(* Logix 5000 project; controller BTS01 vendor 1 type 14 code 217 rev 32.14; software revision 32.04; part 14 of 15 *)
(* tags used below, declared in another part *)
   AG1101 : DTE_VFD;   // Tank 1100 Agitator
   AG1101_CIP_ENABLE : BOOL;
   AG1101_ONS : DINT;
   AG1201 : DTE_VFD;   // Tank 1200 Agitator
   AG1201_CIP_ENABLE : BOOL;
   AG1201_ONS : DINT;
   AirblowPB : BOOL;
   C02S01 : REAL[8];   // 5069-IF8
   C02S02 : REAL[8];   // 5069-OF8
   C02S03 : INT;   // 5069-IB16
   C02S05 : INT;   // 5069-OB16
   C02S06 : INT;   // 5069-IB16
   CIP_1_ACTIVE_CIRCUIT : DINT;
   CIP_1_CIRCUIT_SELECT_HMI : INT;
   CIP_1_RUN_LATCH : BOOL;
   CIP_1_SEQ_CTU : COUNTER;   // CIP 1 SEQUENCE STEP COUNTER THIS IS THE SEQUENCE STEP CONTROL
   CIP_Circuit_1_Visibility : BOOL;
   CIP_Circuit_2_Visibility : BOOL;
   CIP_Circuit_3_Visibility : BOOL;
   CIP_Circuit_4_Visibility : BOOL;
   CIP_SUPPLY_PUMP_CIP_ENABLE : BOOL;
   FP1000_CIP_Supply_Ind : DINT;
   FP1001_CIP_Return_Ind : DINT;
   GlobalAlmAck : BOOL;
   HMIAlarms : DINT[25];   // Alarm Trigger Array
   ONS : DINT[20];   // ONE_SHOT_BIT
   P1001 : DTE_VFD;   // Dressing Tank Fill Pump
   P1001_CIP_Enable : BOOL;
   P1001_ONS : DINT;
   P1001_Start_Request : BOOL;
   P1002 : DTE_VFD;   // Product Filler Fill Pump
   P1002_CIP_ENABLE : BOOL;
   P1002_ONS : DINT;
   P1003 : DTE_VFD;   // CIP Return Pump
   P1003_CIP_ENABLE : BOOL;
   P1003_ONS : DINT;
   P1003_Start_Delay_TMR1 : TIMER;   // CIP Return Pump Active CIP Circuit 1 Start Delay Timer
   P1003_Start_Delay_TMR2 : TIMER;   // CIP Return Pump Active CIP Circuit 2 Start Delay Timer
   P1004 : DTE_VFD;   // Filler CIP Return Pump
   P1004_ONS : DINT;
   TransferEnabled : BOOL;
   TransferSelected : DINT;
   TransferSelection : DINT;
   TransferStandby : BOOL;
   TransferStartPB : BOOL;
   TransferStartPBTimer : TIMER;
   TransferStartPBVisibility : BOOL;
   TransferStopPB : BOOL;
   UnloadEnabled : BOOL;
   UnloadSelected : DINT;
   UnloadSelection : DINT;
   UnloadStandby : BOOL;
   UnloadStartPB : BOOL;
   UnloadStartPBTimer : TIMER;
   UnloadStartPBVisibility : BOOL;
   UnloadStopPB : BOOL;
   V1101 : DTE_Air_Valve_v2;   // Tank 1100 Fill Valve
   V1201 : DTE_Air_Valve_v2;   // Tank 1200 Fill Valve
   ZS1000_1_Ind : DINT;
   ZS1000_2_Ind : DINT;
   ZS1000_3_Ind : DINT;
   ZS1000_4_Ind : DINT;
   ZS1000_5_Ind : DINT;
   ZS1001_1_Ind : DINT;
   ZS1001_2_Ind : DINT;
   ZS1001_3_Ind : DINT;
   ZS1001_4_Ind : DINT;
   ZS1001_5_Ind : DINT;
   ZS1101_Ind : DINT;
   ZS1201_Ind : DINT;
(* MainProgram, continued *)

ROUTINE R06_Motors   (* ladder *)
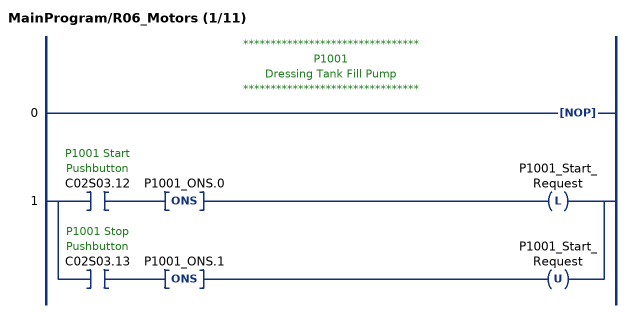
   // ********************************
   // P1001
   // Dressing Tank Fill Pump
   // ********************************
   0: NOP();
   1: [XIC(C02S03.12) ONS(P1001_ONS.0) OTL(P1001_Start_Request) ,XIC(C02S03.13) ONS(P1001_ONS.1) OTU(P1001_Start_Request) ];
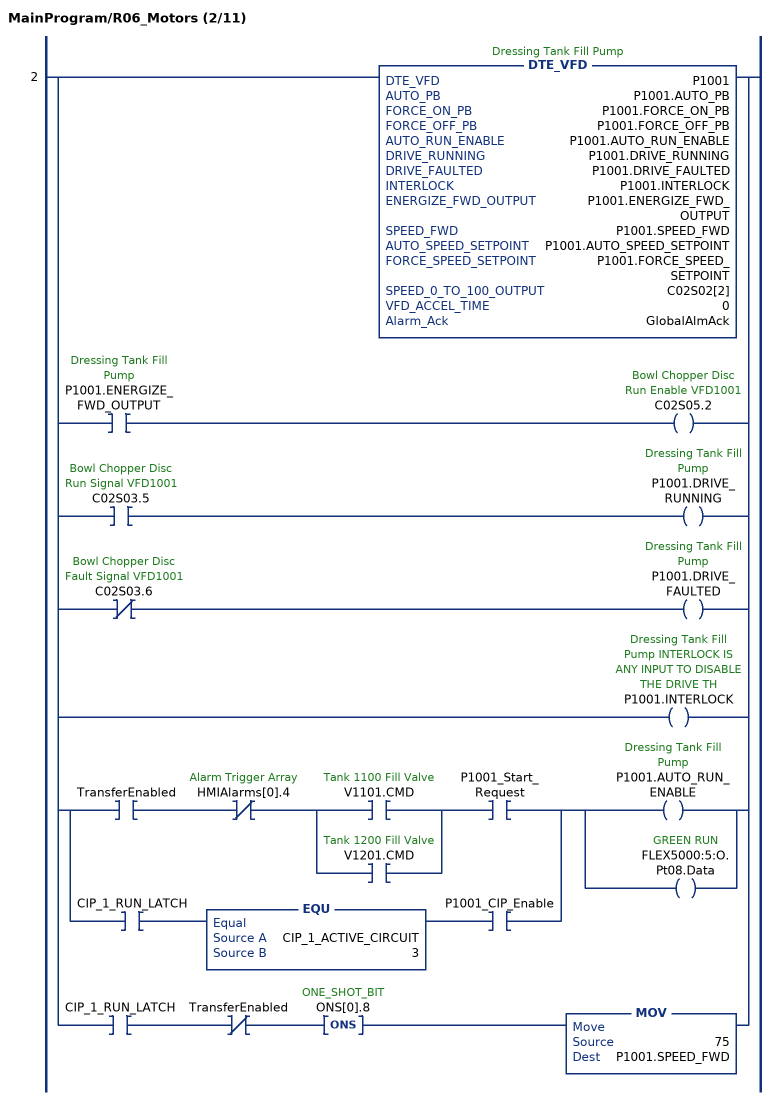
   2: [DTE_VFD(P1001,P1001.AUTO_PB,P1001.FORCE_ON_PB,P1001.FORCE_OFF_PB,P1001.AUTO_RUN_ENABLE,P1001.DRIVE_RUNNING,P1001.DRIVE_FAULTED,P1001.INTERLOCK,P1001.ENERGIZE_FWD_OUTPUT,P1001.SPEED_FWD,P1001.AUTO_SPEED_SETPOINT,P1001.FORCE_SPEED_SETPOINT,C02S02[2],0,GlobalAlmAck) ,XIC(P1001.ENERGIZE_FWD_OUTPUT) OTE(C02S05.2) ,XIC(C02S03.5) OTE(P1001.DRIVE_RUNNING) ,XIO(C02S03.6) OTE(P1001.DRIVE_FAULTED) ,OTE(P1001.INTERLOCK) ,[XIC(TransferEnabled) XIO(HMIAlarms[0].4) [XIC(V1101.CMD) ,XIC(V1201.CMD) ] XIC(P1001_Start_Request) ,XIC(CIP_1_RUN_LATCH) EQU(CIP_1_ACTIVE_CIRCUIT,3) XIC(P1001_CIP_Enable) ] [OTE(P1001.AUTO_RUN_ENABLE) ,OTE(FLEX5000:5:O.Pt08.Data) ] ,XIC(CIP_1_RUN_LATCH) XIO(TransferEnabled) ONS(ONS[0].8) MOV(75,P1001.SPEED_FWD) ];
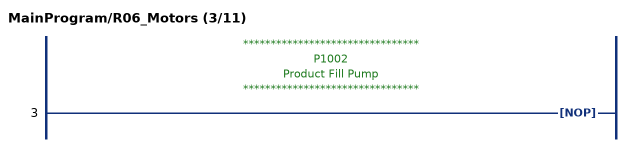
   // ********************************
   // P1002
   // Product Fill Pump
   // ********************************
   3: NOP();
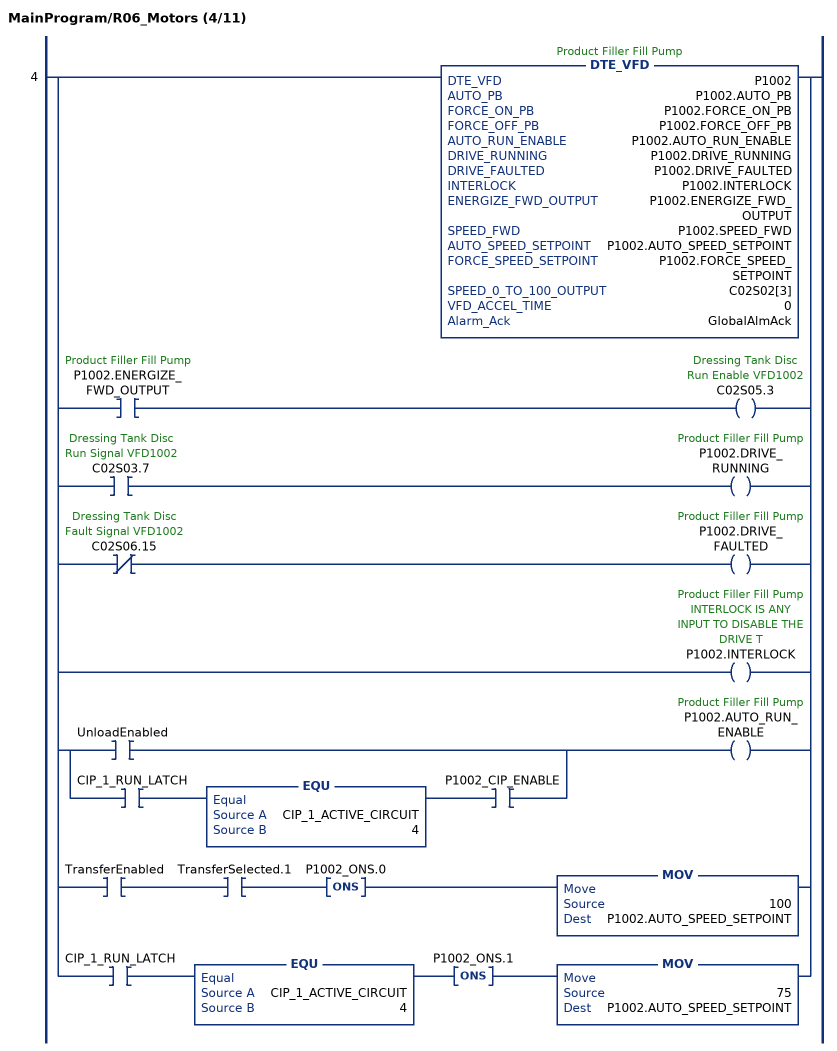
   4: [DTE_VFD(P1002,P1002.AUTO_PB,P1002.FORCE_ON_PB,P1002.FORCE_OFF_PB,P1002.AUTO_RUN_ENABLE,P1002.DRIVE_RUNNING,P1002.DRIVE_FAULTED,P1002.INTERLOCK,P1002.ENERGIZE_FWD_OUTPUT,P1002.SPEED_FWD,P1002.AUTO_SPEED_SETPOINT,P1002.FORCE_SPEED_SETPOINT,C02S02[3],0,GlobalAlmAck) ,XIC(P1002.ENERGIZE_FWD_OUTPUT) OTE(C02S05.3) ,XIC(C02S03.7) OTE(P1002.DRIVE_RUNNING) ,XIO(C02S06.15) OTE(P1002.DRIVE_FAULTED) ,OTE(P1002.INTERLOCK) ,[XIC(UnloadEnabled) ,XIC(CIP_1_RUN_LATCH) EQU(CIP_1_ACTIVE_CIRCUIT,4) XIC(P1002_CIP_ENABLE) ] OTE(P1002.AUTO_RUN_ENABLE) ,XIC(TransferEnabled) XIC(TransferSelected.1) ONS(P1002_ONS.0) MOV(100,P1002.AUTO_SPEED_SETPOINT) ,XIC(CIP_1_RUN_LATCH) EQU(CIP_1_ACTIVE_CIRCUIT,4) ONS(P1002_ONS.1) MOV(75,P1002.AUTO_SPEED_SETPOINT) ];
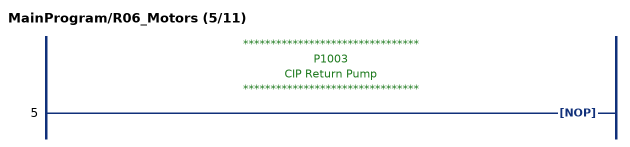
   // ********************************
   // P1003
   // CIP Return Pump
   // ********************************
   5: NOP();
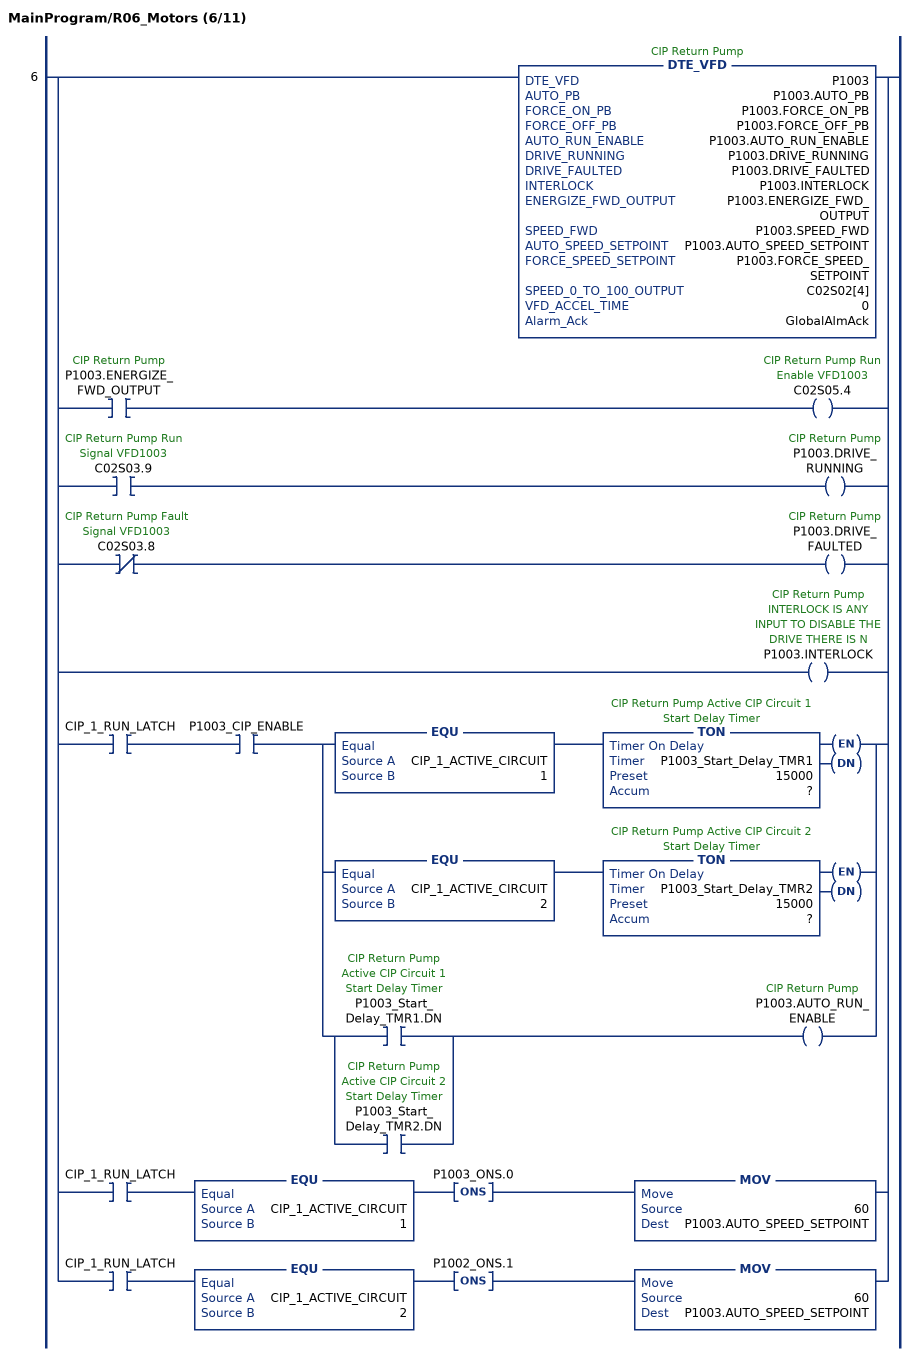
   6: [DTE_VFD(P1003,P1003.AUTO_PB,P1003.FORCE_ON_PB,P1003.FORCE_OFF_PB,P1003.AUTO_RUN_ENABLE,P1003.DRIVE_RUNNING,P1003.DRIVE_FAULTED,P1003.INTERLOCK,P1003.ENERGIZE_FWD_OUTPUT,P1003.SPEED_FWD,P1003.AUTO_SPEED_SETPOINT,P1003.FORCE_SPEED_SETPOINT,C02S02[4],0,GlobalAlmAck) ,XIC(P1003.ENERGIZE_FWD_OUTPUT) OTE(C02S05.4) ,XIC(C02S03.9) OTE(P1003.DRIVE_RUNNING) ,XIO(C02S03.8) OTE(P1003.DRIVE_FAULTED) ,OTE(P1003.INTERLOCK) ,XIC(CIP_1_RUN_LATCH) XIC(P1003_CIP_ENABLE) [EQU(CIP_1_ACTIVE_CIRCUIT,1) TON(P1003_Start_Delay_TMR1,?,?) ,EQU(CIP_1_ACTIVE_CIRCUIT,2) TON(P1003_Start_Delay_TMR2,?,?) ,[XIC(P1003_Start_Delay_TMR1.DN) ,XIC(P1003_Start_Delay_TMR2.DN) ] OTE(P1003.AUTO_RUN_ENABLE) ] ,XIC(CIP_1_RUN_LATCH) EQU(CIP_1_ACTIVE_CIRCUIT,1) ONS(P1003_ONS.0) MOV(60,P1003.AUTO_SPEED_SETPOINT) ,XIC(CIP_1_RUN_LATCH) EQU(CIP_1_ACTIVE_CIRCUIT,2) ONS(P1002_ONS.1) MOV(60,P1003.AUTO_SPEED_SETPOINT) ];
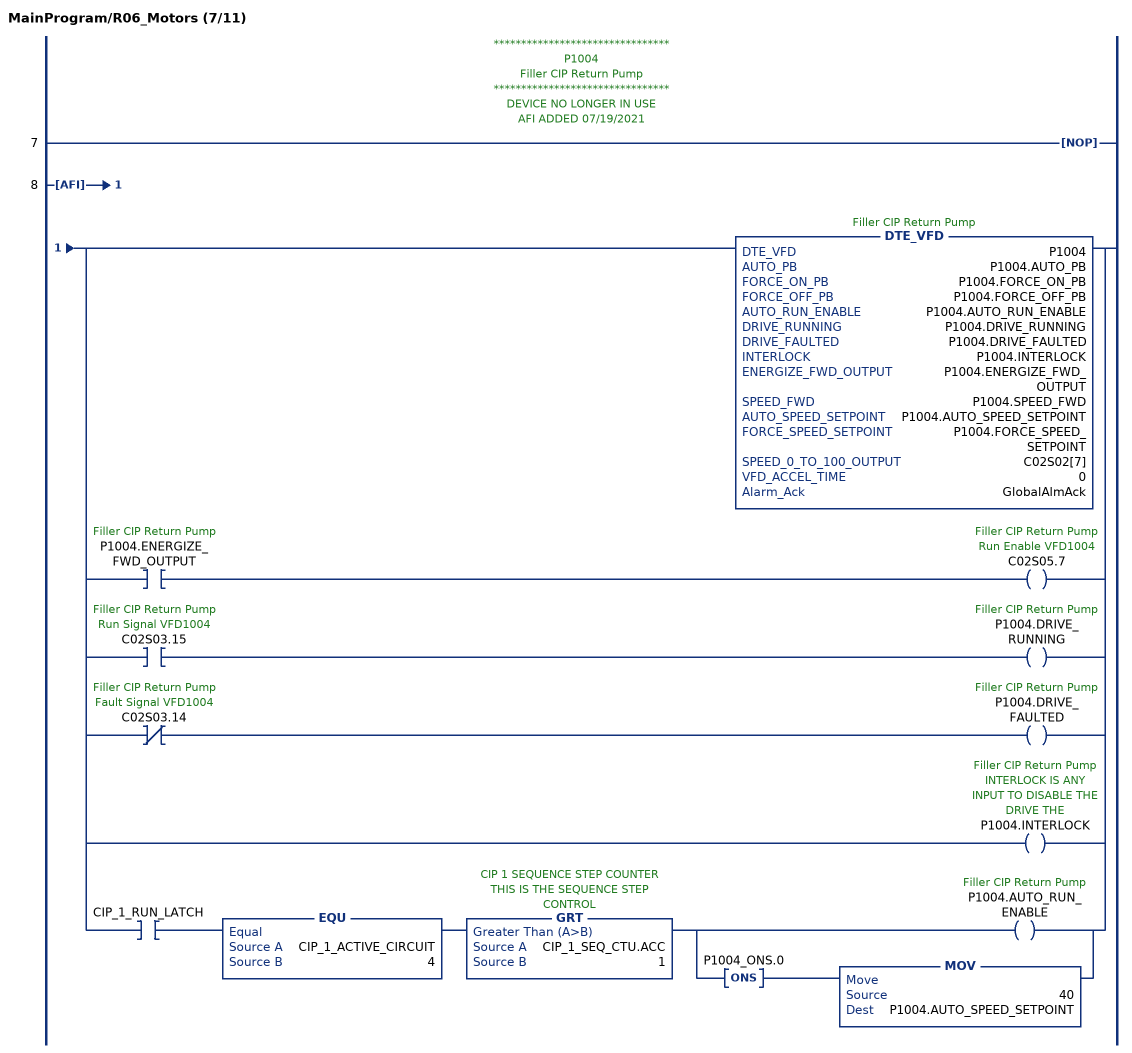
   // ********************************
   // P1004
   // Filler CIP Return Pump
   // ********************************
   // DEVICE NO LONGER IN USE
   // AFI ADDED 07/19/2021
   7: NOP();
   8: AFI()[DTE_VFD(P1004,P1004.AUTO_PB,P1004.FORCE_ON_PB,P1004.FORCE_OFF_PB,P1004.AUTO_RUN_ENABLE,P1004.DRIVE_RUNNING,P1004.DRIVE_FAULTED,P1004.INTERLOCK,P1004.ENERGIZE_FWD_OUTPUT,P1004.SPEED_FWD,P1004.AUTO_SPEED_SETPOINT,P1004.FORCE_SPEED_SETPOINT,C02S02[7],0,GlobalAlmAck) ,XIC(P1004.ENERGIZE_FWD_OUTPUT) OTE(C02S05.7) ,XIC(C02S03.15) OTE(P1004.DRIVE_RUNNING) ,XIO(C02S03.14) OTE(P1004.DRIVE_FAULTED) ,OTE(P1004.INTERLOCK) ,XIC(CIP_1_RUN_LATCH) EQU(CIP_1_ACTIVE_CIRCUIT,4) GRT(CIP_1_SEQ_CTU.ACC,1) [OTE(P1004.AUTO_RUN_ENABLE) ,ONS(P1004_ONS.0) MOV(40,P1004.AUTO_SPEED_SETPOINT) ] ];
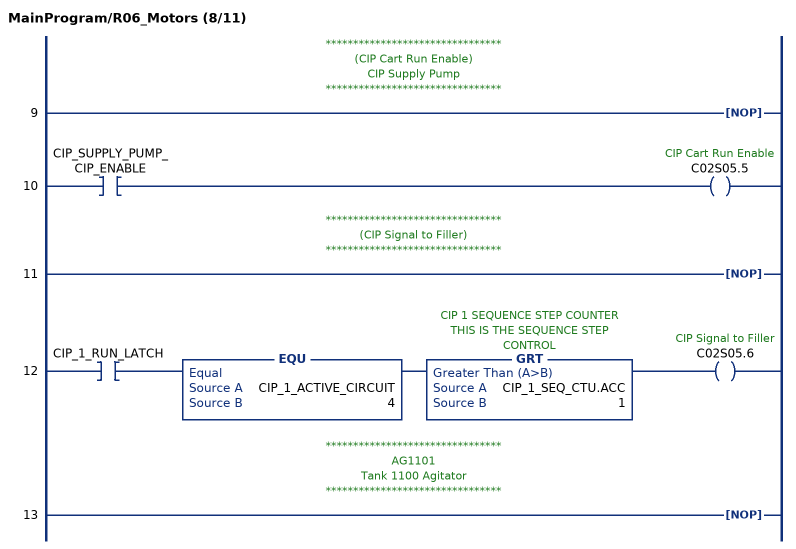
   // ********************************
   // (CIP Cart Run Enable)
   // CIP Supply Pump
   // ********************************
   9: NOP();
   10: XIC(CIP_SUPPLY_PUMP_CIP_ENABLE)OTE(C02S05.5);
   // ********************************
   // (CIP Signal to Filler)
   // ********************************
   11: NOP();
   12: XIC(CIP_1_RUN_LATCH)EQU(CIP_1_ACTIVE_CIRCUIT,4)GRT(CIP_1_SEQ_CTU.ACC,1)OTE(C02S05.6);
   // ********************************
   // AG1101
   // Tank 1100 Agitator
   // ********************************
   13: NOP();
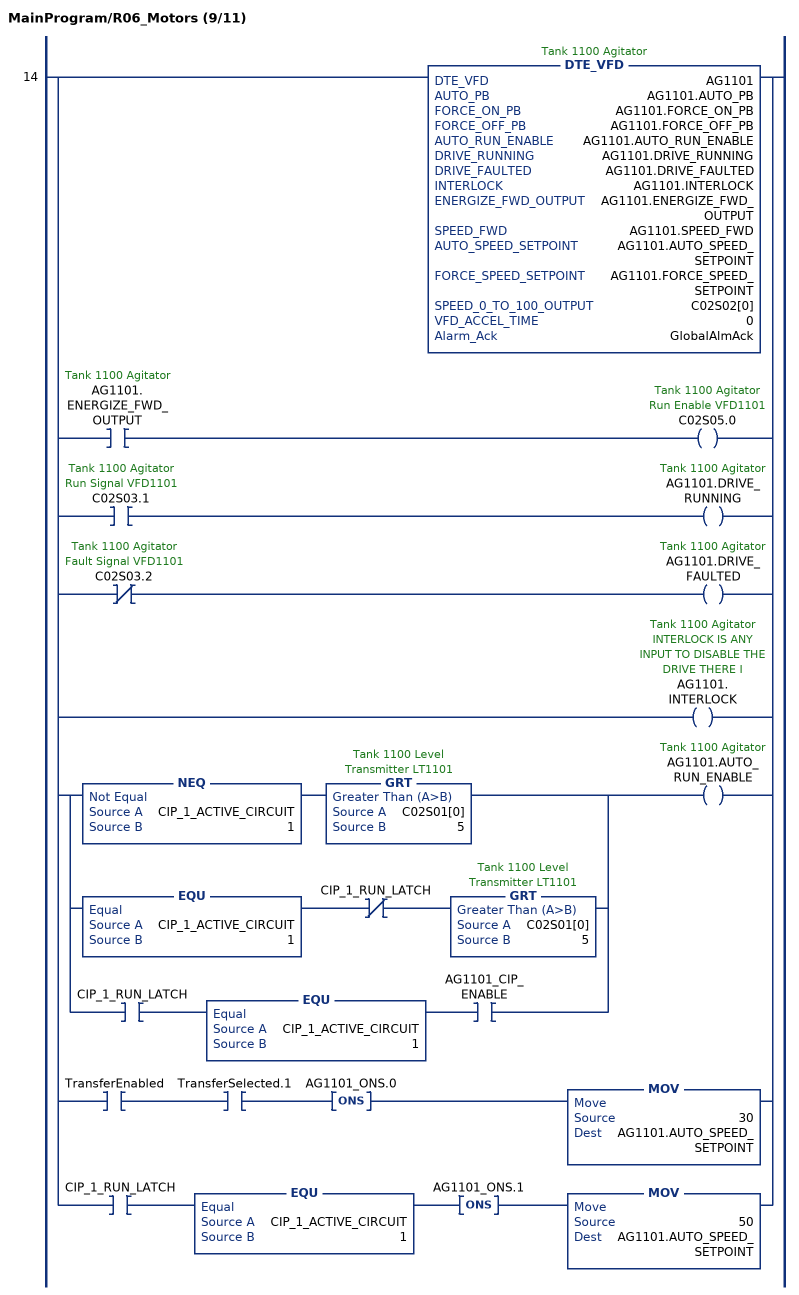
   14: [DTE_VFD(AG1101,AG1101.AUTO_PB,AG1101.FORCE_ON_PB,AG1101.FORCE_OFF_PB,AG1101.AUTO_RUN_ENABLE,AG1101.DRIVE_RUNNING,AG1101.DRIVE_FAULTED,AG1101.INTERLOCK,AG1101.ENERGIZE_FWD_OUTPUT,AG1101.SPEED_FWD,AG1101.AUTO_SPEED_SETPOINT,AG1101.FORCE_SPEED_SETPOINT,C02S02[0],0,GlobalAlmAck) ,XIC(AG1101.ENERGIZE_FWD_OUTPUT) OTE(C02S05.0) ,XIC(C02S03.1) OTE(AG1101.DRIVE_RUNNING) ,XIO(C02S03.2) OTE(AG1101.DRIVE_FAULTED) ,OTE(AG1101.INTERLOCK) ,[NEQ(CIP_1_ACTIVE_CIRCUIT,1) GRT(C02S01[0],5) ,EQU(CIP_1_ACTIVE_CIRCUIT,1) XIO(CIP_1_RUN_LATCH) GRT(C02S01[0],5) ,XIC(CIP_1_RUN_LATCH) EQU(CIP_1_ACTIVE_CIRCUIT,1) XIC(AG1101_CIP_ENABLE) ] OTE(AG1101.AUTO_RUN_ENABLE) ,XIC(TransferEnabled) XIC(TransferSelected.1) ONS(AG1101_ONS.0) MOV(30,AG1101.AUTO_SPEED_SETPOINT) ,XIC(CIP_1_RUN_LATCH) EQU(CIP_1_ACTIVE_CIRCUIT,1) ONS(AG1101_ONS.1) MOV(50,AG1101.AUTO_SPEED_SETPOINT) ];
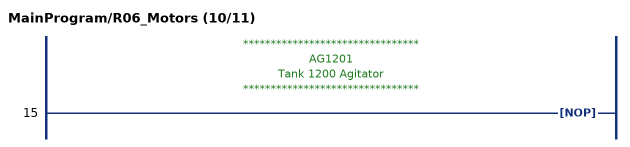
   // ********************************
   // AG1201
   // Tank 1200 Agitator
   // ********************************
   15: NOP();
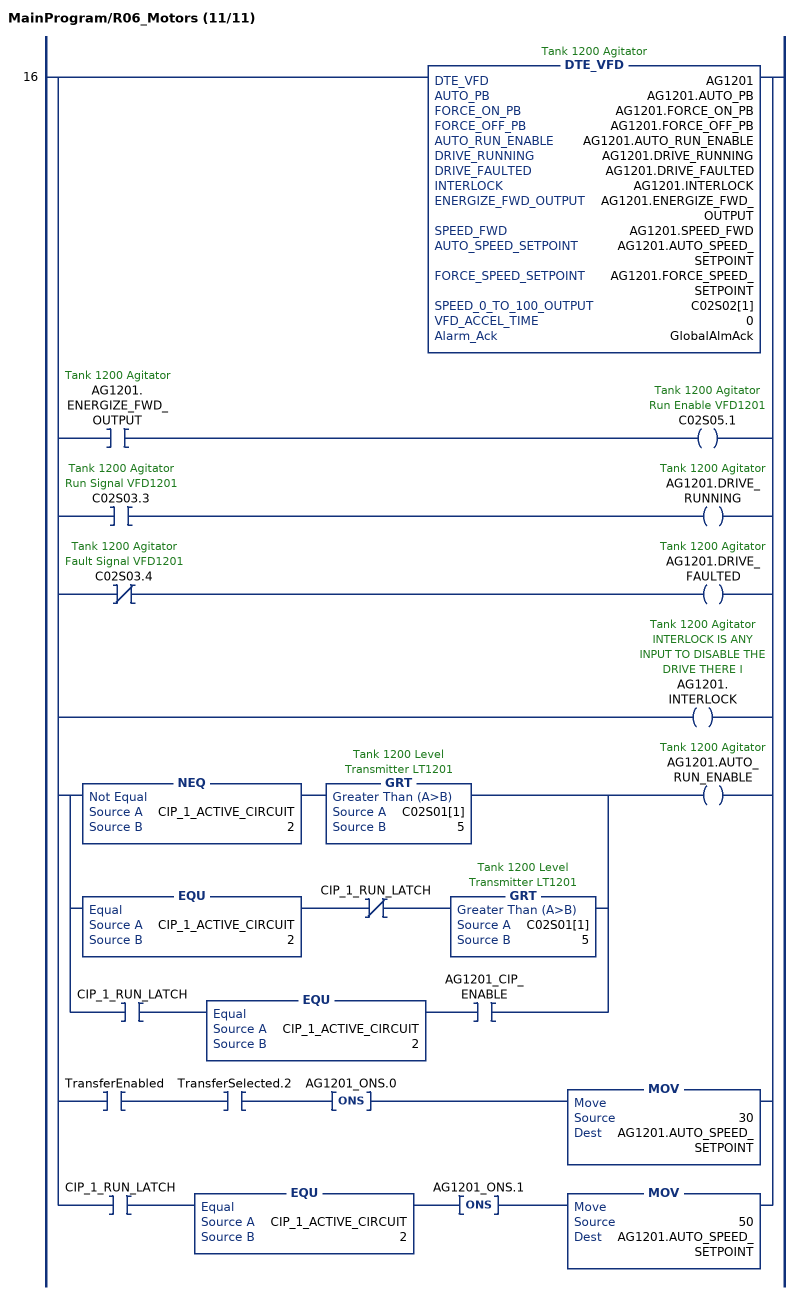
   16: [DTE_VFD(AG1201,AG1201.AUTO_PB,AG1201.FORCE_ON_PB,AG1201.FORCE_OFF_PB,AG1201.AUTO_RUN_ENABLE,AG1201.DRIVE_RUNNING,AG1201.DRIVE_FAULTED,AG1201.INTERLOCK,AG1201.ENERGIZE_FWD_OUTPUT,AG1201.SPEED_FWD,AG1201.AUTO_SPEED_SETPOINT,AG1201.FORCE_SPEED_SETPOINT,C02S02[1],0,GlobalAlmAck) ,XIC(AG1201.ENERGIZE_FWD_OUTPUT) OTE(C02S05.1) ,XIC(C02S03.3) OTE(AG1201.DRIVE_RUNNING) ,XIO(C02S03.4) OTE(AG1201.DRIVE_FAULTED) ,OTE(AG1201.INTERLOCK) ,[NEQ(CIP_1_ACTIVE_CIRCUIT,2) GRT(C02S01[1],5) ,EQU(CIP_1_ACTIVE_CIRCUIT,2) XIO(CIP_1_RUN_LATCH) GRT(C02S01[1],5) ,XIC(CIP_1_RUN_LATCH) EQU(CIP_1_ACTIVE_CIRCUIT,2) XIC(AG1201_CIP_ENABLE) ] OTE(AG1201.AUTO_RUN_ENABLE) ,XIC(TransferEnabled) XIC(TransferSelected.2) ONS(AG1201_ONS.0) MOV(30,AG1201.AUTO_SPEED_SETPOINT) ,XIC(CIP_1_RUN_LATCH) EQU(CIP_1_ACTIVE_CIRCUIT,2) ONS(AG1201_ONS.1) MOV(50,AG1201.AUTO_SPEED_SETPOINT) ];
END_ROUTINE

ROUTINE R10_Transfer   (* ladder *)
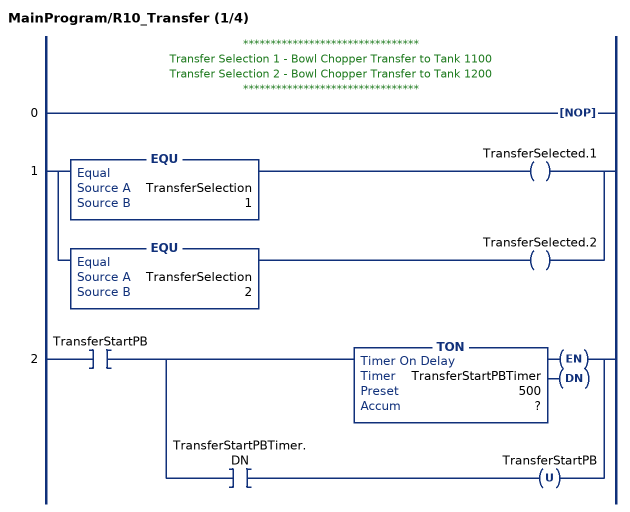
   // ********************************
   // Transfer Selection 1 - Bowl Chopper Transfer to Tank 1100
   // Transfer Selection 2 - Bowl Chopper Transfer to Tank 1200
   // ********************************
   0: NOP();
   1: [EQU(TransferSelection,1) OTE(TransferSelected.1) ,EQU(TransferSelection,2) OTE(TransferSelected.2) ];
   2: XIC(TransferStartPB)[TON(TransferStartPBTimer,?,?) ,XIC(TransferStartPBTimer.DN) OTU(TransferStartPB) ];
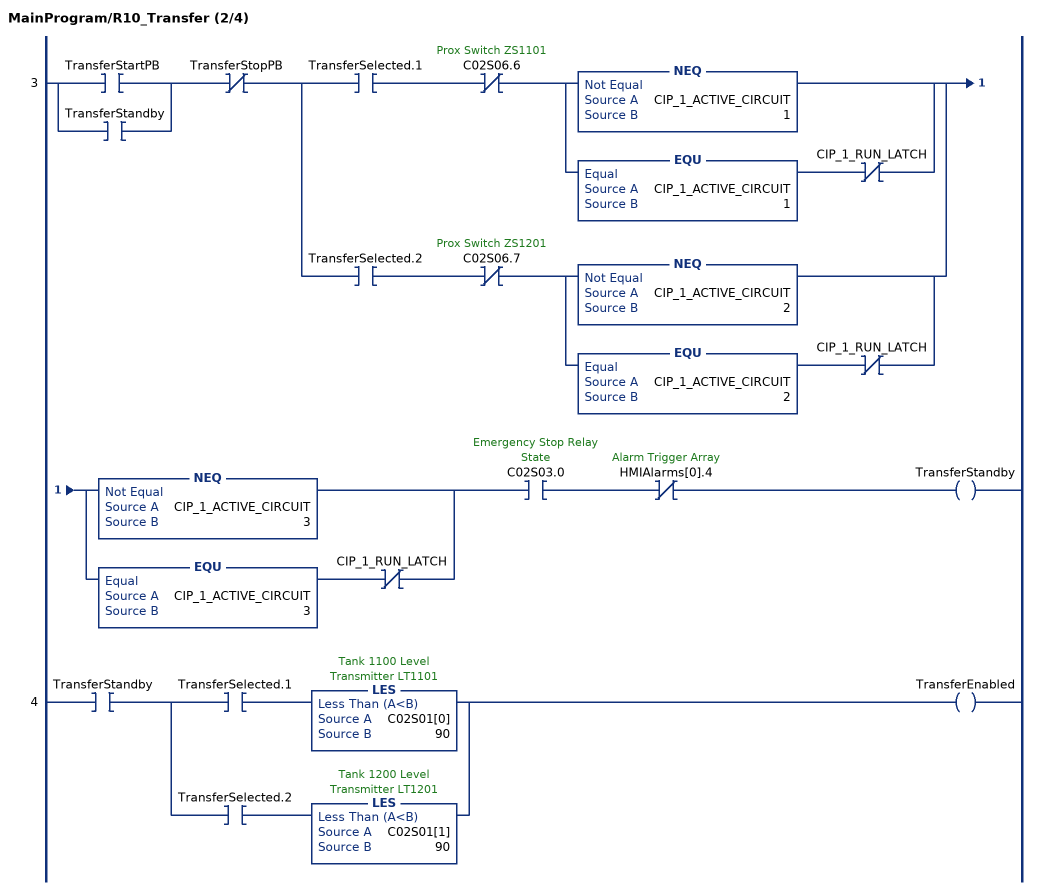
   3: [XIC(TransferStartPB) ,XIC(TransferStandby) ]XIO(TransferStopPB)[XIC(TransferSelected.1) XIO(C02S06.6) [NEQ(CIP_1_ACTIVE_CIRCUIT,1) ,EQU(CIP_1_ACTIVE_CIRCUIT,1) XIO(CIP_1_RUN_LATCH) ] ,XIC(TransferSelected.2) XIO(C02S06.7) [NEQ(CIP_1_ACTIVE_CIRCUIT,2) ,EQU(CIP_1_ACTIVE_CIRCUIT,2) XIO(CIP_1_RUN_LATCH) ] ][NEQ(CIP_1_ACTIVE_CIRCUIT,3) ,EQU(CIP_1_ACTIVE_CIRCUIT,3) XIO(CIP_1_RUN_LATCH) ]XIC(C02S03.0)XIO(HMIAlarms[0].4)OTE(TransferStandby);
   4: XIC(TransferStandby)[XIC(TransferSelected.1) LES(C02S01[0],90) ,XIC(TransferSelected.2) LES(C02S01[1],90) ]OTE(TransferEnabled);
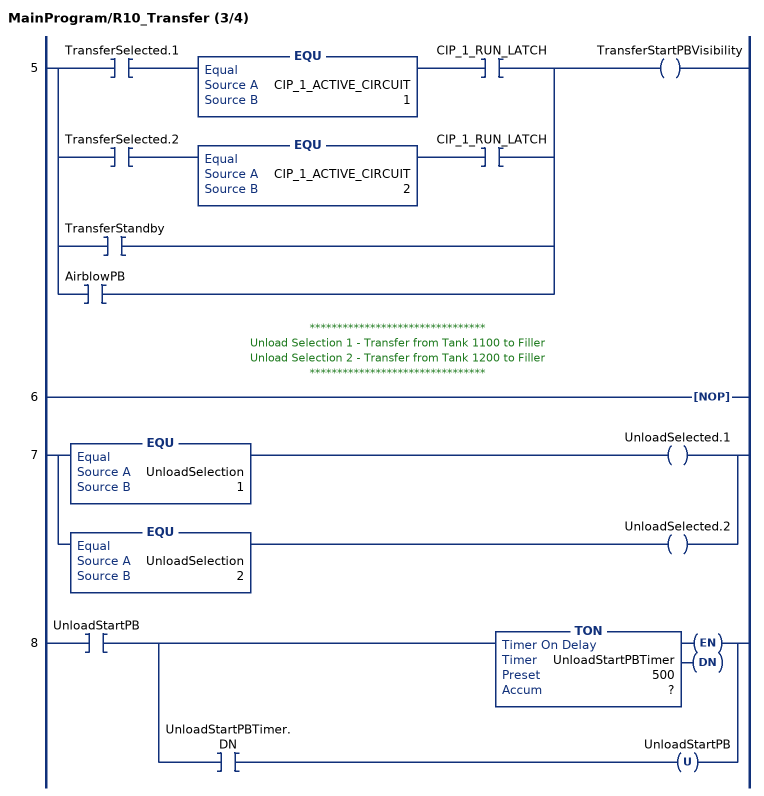
   5: [XIC(TransferSelected.1) EQU(CIP_1_ACTIVE_CIRCUIT,1) XIC(CIP_1_RUN_LATCH) ,XIC(TransferSelected.2) EQU(CIP_1_ACTIVE_CIRCUIT,2) XIC(CIP_1_RUN_LATCH) ,XIC(TransferStandby) ,XIC(AirblowPB) ]OTE(TransferStartPBVisibility);
   // ********************************
   // Unload Selection 1 - Transfer from Tank 1100 to Filler
   // Unload Selection 2 - Transfer from Tank 1200 to Filler
   // ********************************
   6: NOP();
   7: [EQU(UnloadSelection,1) OTE(UnloadSelected.1) ,EQU(UnloadSelection,2) OTE(UnloadSelected.2) ];
   8: XIC(UnloadStartPB)[TON(UnloadStartPBTimer,?,?) ,XIC(UnloadStartPBTimer.DN) OTU(UnloadStartPB) ];
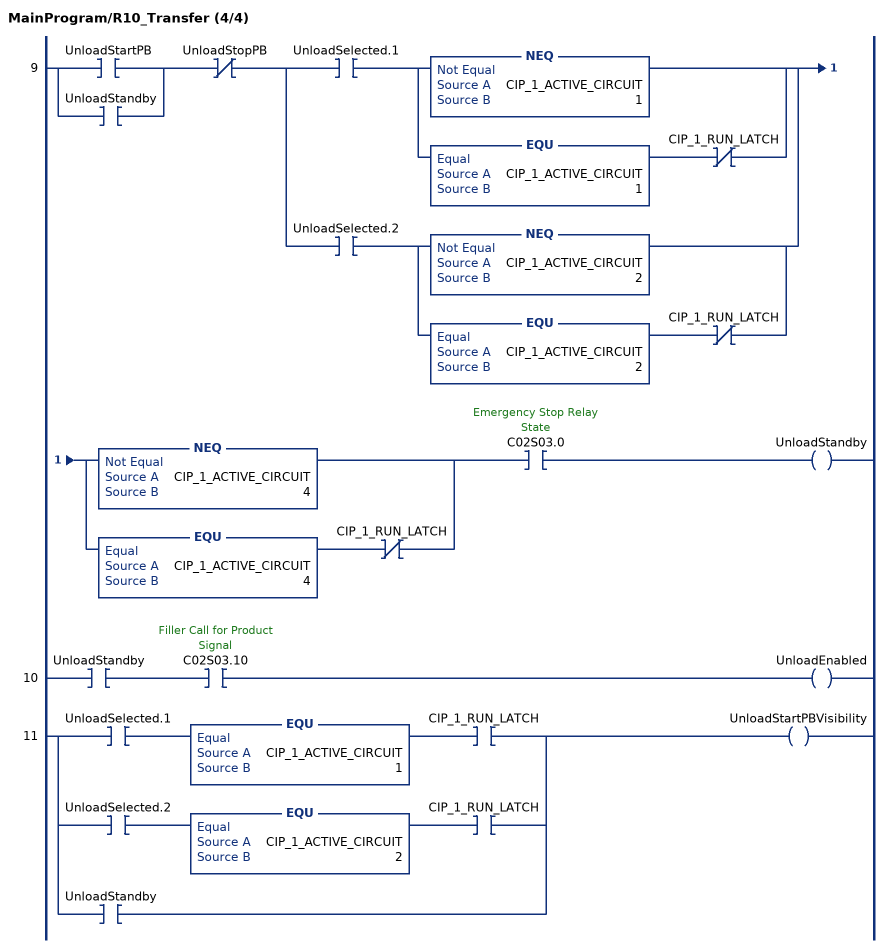
   9: [XIC(UnloadStartPB) ,XIC(UnloadStandby) ]XIO(UnloadStopPB)[XIC(UnloadSelected.1) [NEQ(CIP_1_ACTIVE_CIRCUIT,1) ,EQU(CIP_1_ACTIVE_CIRCUIT,1) XIO(CIP_1_RUN_LATCH) ] ,XIC(UnloadSelected.2) [NEQ(CIP_1_ACTIVE_CIRCUIT,2) ,EQU(CIP_1_ACTIVE_CIRCUIT,2) XIO(CIP_1_RUN_LATCH) ] ][NEQ(CIP_1_ACTIVE_CIRCUIT,4) ,EQU(CIP_1_ACTIVE_CIRCUIT,4) XIO(CIP_1_RUN_LATCH) ]XIC(C02S03.0)OTE(UnloadStandby);
   10: XIC(UnloadStandby)XIC(C02S03.10)OTE(UnloadEnabled);
   11: [XIC(UnloadSelected.1) EQU(CIP_1_ACTIVE_CIRCUIT,1) XIC(CIP_1_RUN_LATCH) ,XIC(UnloadSelected.2) EQU(CIP_1_ACTIVE_CIRCUIT,2) XIC(CIP_1_RUN_LATCH) ,XIC(UnloadStandby) ]OTE(UnloadStartPBVisibility);
END_ROUTINE

ROUTINE R12_Sensor_Interlocks   (* ladder *)
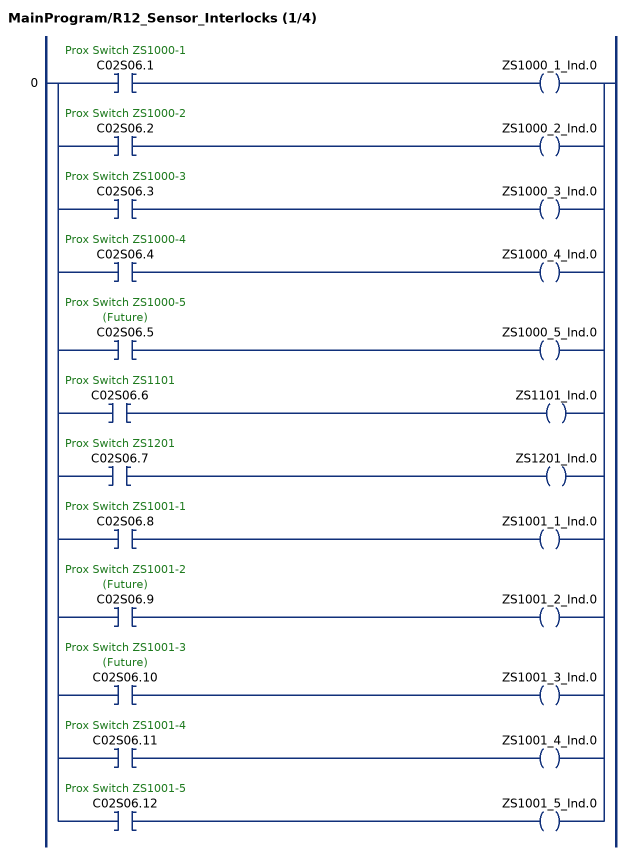
   0: [XIC(C02S06.1) OTE(ZS1000_1_Ind.0) ,XIC(C02S06.2) OTE(ZS1000_2_Ind.0) ,XIC(C02S06.3) OTE(ZS1000_3_Ind.0) ,XIC(C02S06.4) OTE(ZS1000_4_Ind.0) ,XIC(C02S06.5) OTE(ZS1000_5_Ind.0) ,XIC(C02S06.6) OTE(ZS1101_Ind.0) ,XIC(C02S06.7) OTE(ZS1201_Ind.0) ,XIC(C02S06.8) OTE(ZS1001_1_Ind.0) ,XIC(C02S06.9) OTE(ZS1001_2_Ind.0) ,XIC(C02S06.10) OTE(ZS1001_3_Ind.0) ,XIC(C02S06.11) OTE(ZS1001_4_Ind.0) ,XIC(C02S06.12) OTE(ZS1001_5_Ind.0) ];
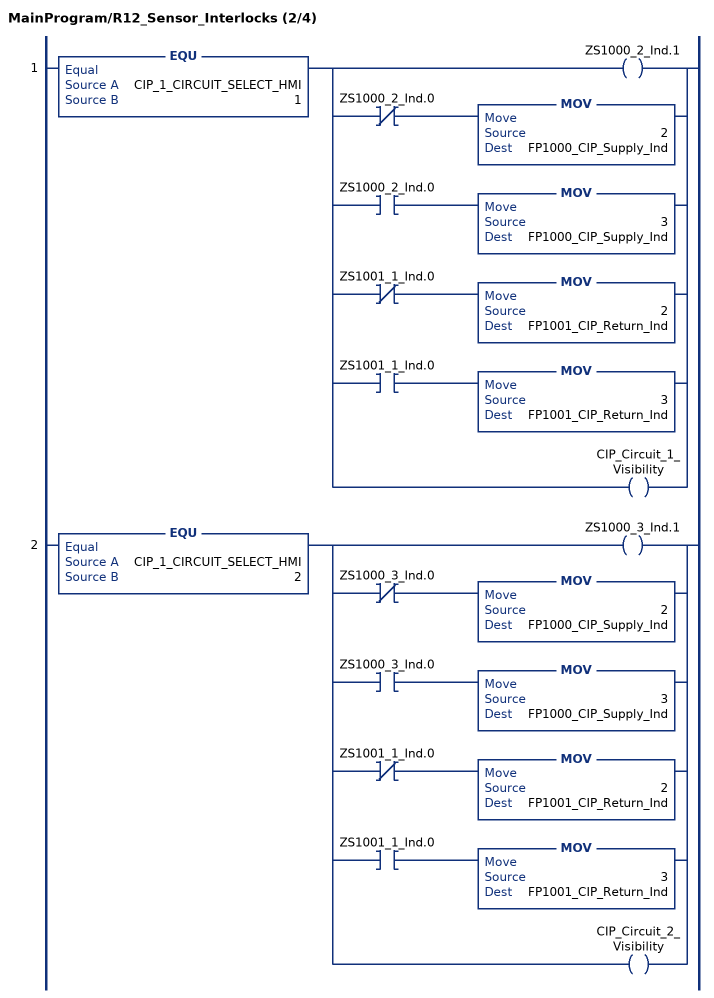
   1: EQU(CIP_1_CIRCUIT_SELECT_HMI,1)[OTE(ZS1000_2_Ind.1) ,XIO(ZS1000_2_Ind.0) MOV(2,FP1000_CIP_Supply_Ind) ,XIC(ZS1000_2_Ind.0) MOV(3,FP1000_CIP_Supply_Ind) ,XIO(ZS1001_1_Ind.0) MOV(2,FP1001_CIP_Return_Ind) ,XIC(ZS1001_1_Ind.0) MOV(3,FP1001_CIP_Return_Ind) ,OTE(CIP_Circuit_1_Visibility) ];
   2: EQU(CIP_1_CIRCUIT_SELECT_HMI,2)[OTE(ZS1000_3_Ind.1) ,XIO(ZS1000_3_Ind.0) MOV(2,FP1000_CIP_Supply_Ind) ,XIC(ZS1000_3_Ind.0) MOV(3,FP1000_CIP_Supply_Ind) ,XIO(ZS1001_1_Ind.0) MOV(2,FP1001_CIP_Return_Ind) ,XIC(ZS1001_1_Ind.0) MOV(3,FP1001_CIP_Return_Ind) ,OTE(CIP_Circuit_2_Visibility) ];
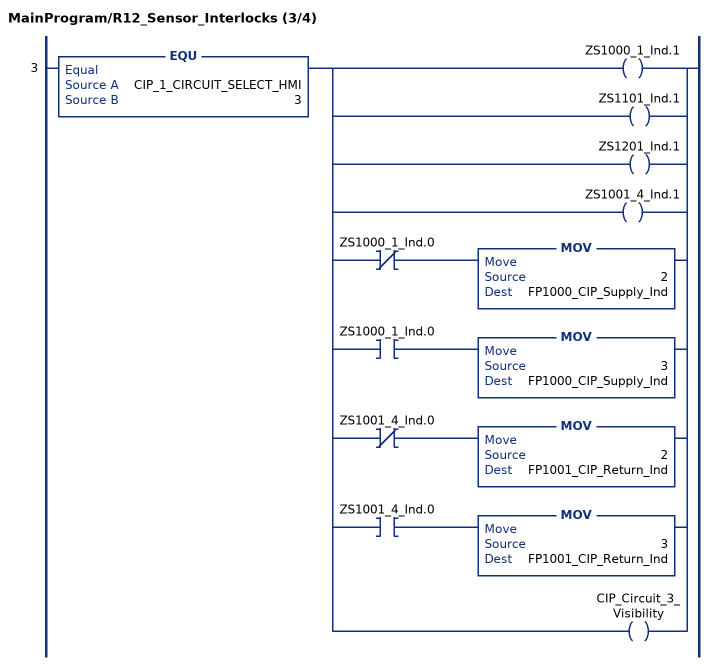
   3: EQU(CIP_1_CIRCUIT_SELECT_HMI,3)[OTE(ZS1000_1_Ind.1) ,OTE(ZS1101_Ind.1) ,OTE(ZS1201_Ind.1) ,OTE(ZS1001_4_Ind.1) ,XIO(ZS1000_1_Ind.0) MOV(2,FP1000_CIP_Supply_Ind) ,XIC(ZS1000_1_Ind.0) MOV(3,FP1000_CIP_Supply_Ind) ,XIO(ZS1001_4_Ind.0) MOV(2,FP1001_CIP_Return_Ind) ,XIC(ZS1001_4_Ind.0) MOV(3,FP1001_CIP_Return_Ind) ,OTE(CIP_Circuit_3_Visibility) ];
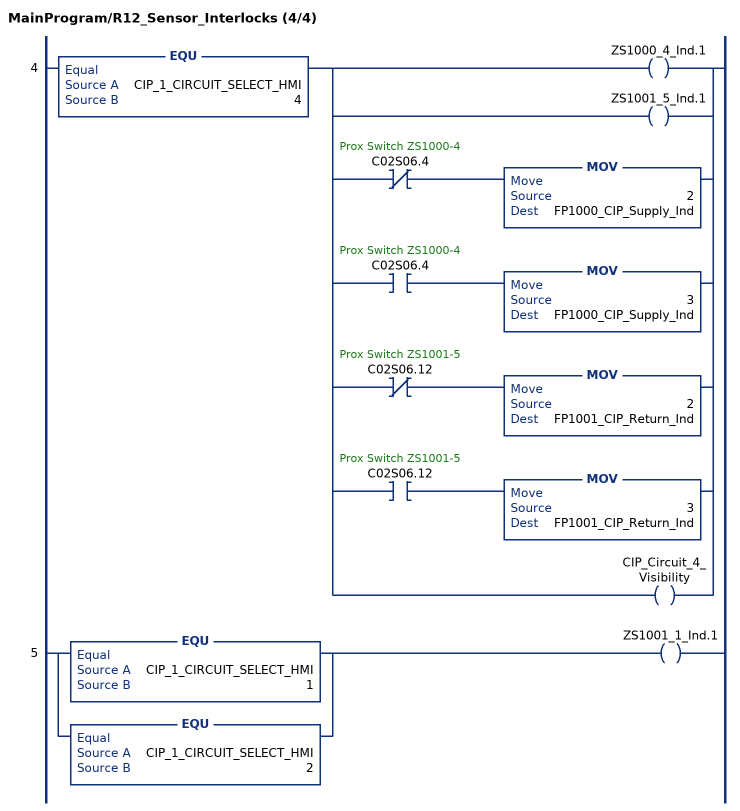
   4: EQU(CIP_1_CIRCUIT_SELECT_HMI,4)[OTE(ZS1000_4_Ind.1) ,OTE(ZS1001_5_Ind.1) ,XIO(C02S06.4) MOV(2,FP1000_CIP_Supply_Ind) ,XIC(C02S06.4) MOV(3,FP1000_CIP_Supply_Ind) ,XIO(C02S06.12) MOV(2,FP1001_CIP_Return_Ind) ,XIC(C02S06.12) MOV(3,FP1001_CIP_Return_Ind) ,OTE(CIP_Circuit_4_Visibility) ];
   5: [EQU(CIP_1_CIRCUIT_SELECT_HMI,1) ,EQU(CIP_1_CIRCUIT_SELECT_HMI,2) ]OTE(ZS1001_1_Ind.1);
END_ROUTINE
